// TIA Portal V20 export
TYPE "typeCmControlNodeCommand"
// stored: Namespace Unit1.Em5
   STRUCT
      transferPnPLeftAxisX : "LER_typeAxisCommand";
      transferPnPLeftAxisY : "LER_typeAxisCommand";
      transferPnPLeftAxisZ { S7_SetPoint := 'True'} : "LER_typeAxisCommand";
      transferPnPRightAxisX { S7_SetPoint := 'True'} : "LER_typeAxisCommand";
      transferPnPRightAxisY { S7_SetPoint := 'True'} : "LER_typeAxisCommand";
      transferPnPRightAxisZ { S7_SetPoint := 'True'} : "LER_typeAxisCommand";
      transferPnPLeftClamp { S7_SetPoint := 'True'} : "LER_typeTwoWayActCommand";
      transferPnPRightClamp { S7_SetPoint := 'True'} : "LER_typeTwoWayActCommand";
   END_STRUCT;
END_TYPE
